TYPE SmokeControlFireParameters :
STRUCT
	EN: BOOL := TRUE;
END_STRUCT
END_TYPE

(* stored: Version 1.1.0.1, ProductVersion 3.1.4024.6
   DUT SmokeControlFireParameters: Id {beb37f6f-2c07-4ee8-a55d-164b4697df20} *)
